FUNCTION_BLOCK TcoLoggerEnrichmentConfiguration

VAR_INPUT
	Config		: REFERENCE TO TcoLoggerConfiguration;
END_VAR

VAR
	_instancePathEnricher 	: InstancePathEnricher;
END_VAR

METHOD PUBLIC Context : REFERENCE TO TcoLoggerConfiguration
VAR_INPUT
END_VAR
Context REF= Config;
END_METHOD

METHOD PUBLIC CycleCount : REFERENCE TO TcoLoggerConfiguration
VAR_INPUT
END_VAR
CycleCount REF= Config;
END_METHOD

METHOD PUBLIC InstancePath : REFERENCE TO TcoLoggerConfiguration
VAR_INPUT
END_VAR
Config.AddEnrichment(_instancePathEnricher);
InstancePath REF= Config;
END_METHOD

END_FUNCTION_BLOCK

(* stored: Version 1.1.0.1, ProductVersion 3.1.4024.9
   POU TcoLoggerEnrichmentConfiguration: Id {41bdeba9-659c-0092-3e34-84293c8dbc97}, SpecialFunc None
   Method Context: Id {755538a3-16a8-0e8a-16e4-53fad2283699}
   Method CycleCount: Id {0a423684-22e3-0e09-347c-52c7bcc3a745}
   Method InstancePath: Id {2a11cc84-95b7-0afc-3082-caec0b84ec93} *)
